// TIA Portal V17 export
// export: Created 2022-07-20T06:59:34.3263175Z, ExportSetting WithDefaults, DisplayName Totally Integrated Automation Portal, DisplayVersion V17, DisplayName TIA Portal Openness, DisplayVersion V17, DisplayName TIA Portal Version Control Interface, DisplayVersion V17, DisplayName SINAMICS Startdrive Advanced, DisplayVersion V17, DisplayName SINAMICS Startdrive G130, G150, S120, S150, SINAMICS MV, S210, DisplayVersion V17, DisplayName SINAMICS Startdrive G110M, G120, G120C, G120D, G120P, G115D, DisplayVersion V17, DisplayName STEP 7 Professional, DisplayVersion V17, DisplayName STEP 7 Safety, DisplayVersion V17, DisplayName WinCC Advanced, DisplayVersion V17
FUNCTION "FC1_Program_Version_&_Release_Note" : Void   // FC1, LAD
{ S7_Optimized_Access := 'TRUE' }
VERSION : 0.1
// stored: AutoNumber false, IsIECCheckEnabled false, SetENOAutomatically false, UDAEnableTagReadback false
BEGIN

REGION Network 1 (SCL): Programm Version
   "DB_Machine".Version.Major := 0;
   "DB_Machine".Version.Minor := 0;
   "DB_Machine".Version.Patch := 6;
   "DB_Machine".Version.Alpha := TRUE;
   "DB_Machine".Version.Beta  := TRUE;
END_REGION

REGION Network 3 (SCL): TODO
END_REGION

REGION Network 4 (SCL): Version 0.0.7
   (*JONATHAN - 02/05/2022*)
   // [NEW] - Intégration du KP Adaptation pour les winders
   // [NEW] - Ajout des last images des printers P1 et P2
   // [CHANGE] - Prise en compte du front descendant des last images
   //
END_REGION

REGION Network 5 (SCL): Version 0.0.6
   (*JONATHAN - 28/04/2022*)
   // [FIX] - Change config TO PTO pour générer 1 pulse / 10um
   // [NEW] - Ajout du AL2301 pour pilotage du blocage web guide et de l'autorisation de printing à la sync board
   // [CHANGE] - Changement du type de pilotage du PTO pour etre sur Pulse (A) + Sens (B) + changement d'E/S syncoard
END_REGION

REGION Network 6 (SCL): Version 0.0.5
   (*ANIROUDDH - 20/04/2022*)
   // [FIX] - Acknwoledge cablé sur les moteurs
END_REGION
END_FUNCTION
